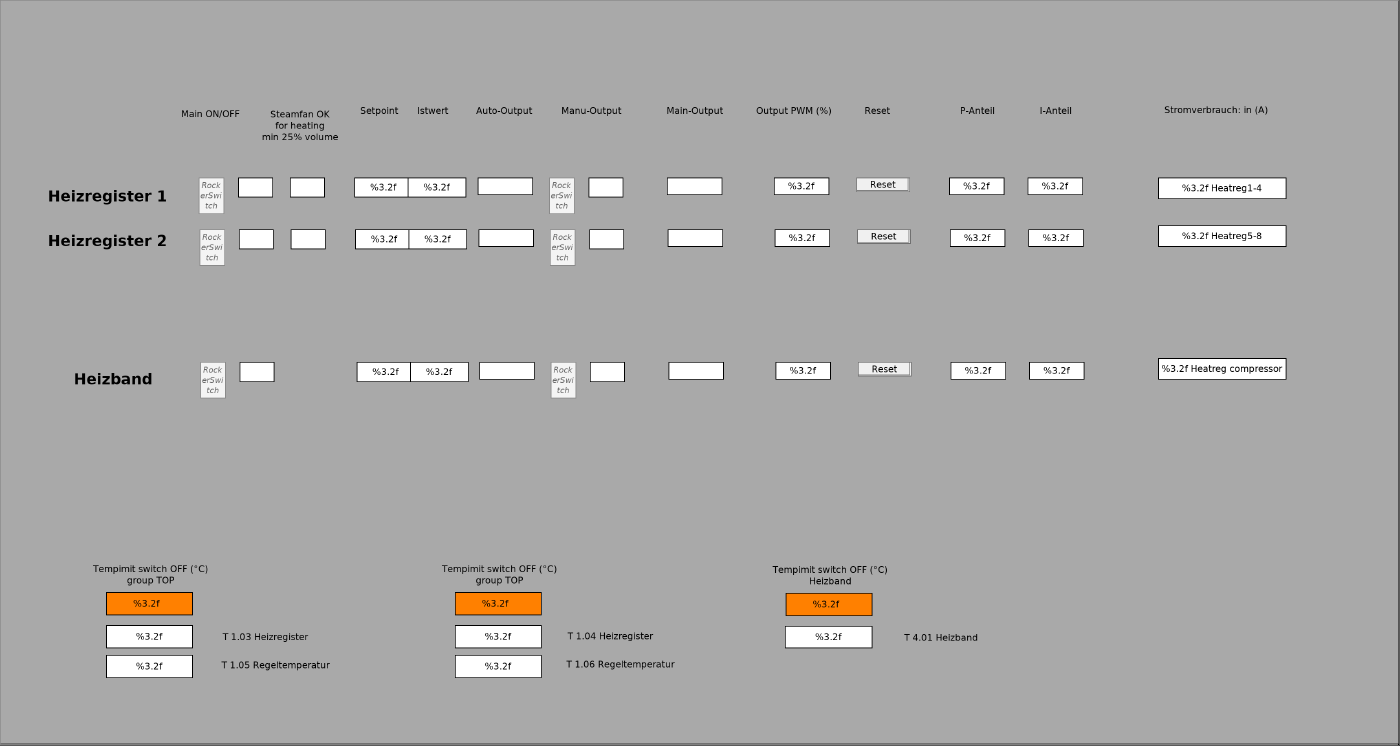
VISUALIZATION Heatreg  // 1782x950
    Rectangle (451,226 74x25), "%3.2f", tooltip "Durchmesser in mm eingeben", text variable: GVL.fSetpointValue1
        OnMouseDown: write the text variable via VisuDialogs.Numpad, min 0, max 150
    Rectangle (596,126 92x30), "Auto-Output"
    Rectangle (707,126 92x30), "Manu-Output"
    Rectangle (839,126 92x30), "Main-Output"
    Rectangle (437,126 92x30), "Setpoint"
    Rectangle (609,292 70x22), colour toggle: GVL.bAuto_Heat_REG2_CTRL
    Rectangle (850,292 70x22), colour toggle: GVL.HEAT_Reg_2_OUT
    Rectangle (608,226 70x22), colour toggle: GVL.bAuto_Heat_REG1_CTRL
    Rectangle (849,226 70x22), colour toggle: GVL.HEAT_Reg_1_OUT
    Rectangle (951,126 116x30), "Output PWM (%)"
    Rectangle (986,292 70x22), "%3.2f", text variable: fPWMDutyCycle2
    Rectangle (985,226 70x22), "%3.2f", text variable: fPWMDutyCycle1
    Rectangle (610,461 70x22), colour toggle: GVL.bAuto_Heat_REG3_CTRL
    Rectangle (851,461 70x22), colour toggle: GVL.HEAT_Reg_3_OUT
    Rectangle (987,461 70x22), "%3.2f", text variable: fPWMDutyCycle3
    Rectangle (1473,124 150x32), "Stromverbrauch: in (A)"
    Rectangle (750,292 44x25), colour toggle: GVL.bManuHeat_REG2_CTRL
    Rectangle (749,226 44x25), colour toggle: GVL.bManuHeat_REG1_CTRL
    Rectangle (751,461 44x25), colour toggle: GVL.bManuHeat_REG3_CTRL
    Rectangle (135,754 110x29), "%3.2f", tooltip "Durchmesser in mm eingeben", text variable: GVL.T_Limit_Heatreg_top
        OnMouseDown: write the text variable via VisuDialogs.Numpad, min 0, max 300
    Rectangle (107,718 170x28), "Tempimit switch OFF (°C) group TOP"
    Rectangle (135,796 110x29), "%3.2f", tooltip "Durchmesser in mm eingeben", text variable: GVL.T_HE_Einduesung_Oben_Visu
    Rectangle (135,834 110x29), "%3.2f", tooltip "Durchmesser in mm eingeben", text variable: GVL.T_Einduesung_Oben_Visu
    Rectangle (265,798 146x26), "T 1.03 Heizregister"
    Rectangle (265,834 172x26), "T 1.05 Regeltemperatur"
    Rectangle (579,754 110x29), "%3.2f", tooltip "Durchmesser in mm eingeben", text variable: GVL.T_Limit_Heatreg_bottom
        OnMouseDown: write the text variable via VisuDialogs.Numpad, min 0, max 300
    Rectangle (551,718 170x28), "Tempimit switch OFF (°C) group TOP"
    Rectangle (579,796 110x29), "%3.2f", tooltip "Durchmesser in mm eingeben", text variable: GVL.T_HE_Einduesung_Unten_Visu
    Rectangle (579,834 110x29), "%3.2f", tooltip "Durchmesser in mm eingeben", text variable: GVL.T_Einduesung_Unten_Visu
    Rectangle (1780,0 2x950)
    Rectangle (0,947 1780x3)
    RockerSwitch (699,226 32x46), variable: GVL.bManuHeat_REG1_CTRL, behaviour: TOGGLE, style: Switch-RockerSwitch-Gray
    RockerSwitch (700,292 32x46), variable: GVL.bManuHeat_REG2_CTRL, behaviour: TOGGLE, style: Switch-RockerSwitch-Gray
    RockerSwitch (701,461 32x46), variable: GVL.bManuHeat_REG3_CTRL, behaviour: TOGGLE, style: Switch-RockerSwitch-Gray
    Rectangle (452,292 74x25), "%3.2f", tooltip "Durchmesser in mm eingeben", text variable: GVL.fSetpointValue2
        OnMouseDown: write the text variable via VisuDialogs.Numpad, min 0, max 150
    Rectangle (454,461 74x25), "%3.2f", tooltip "Durchmesser in mm eingeben", text variable: GVL.fSetpointValue3
        OnMouseDown: write the text variable via VisuDialogs.Numpad, min 0, max 150
    Rectangle (1071,126 92x30), "Reset"
    Button (1092,461 68x18), "Reset"
        tap Reset_heatreg_compressor
    Button (1090,226 68x18), "Reset"
        tap Reset_heatreg_top
    Button (1091,292 68x18), "Reset"
        tap Reset_heatreg_bottom
    Rectangle (370,292 44x25), colour toggle: OK_For_HEAT_WHILE_FAN_IS_ON
    Rectangle (369,226 44x25), colour toggle: OK_For_HEAT_WHILE_FAN_IS_ON
    Rectangle (328,132 108x56), "Steamfan OK for heating min 25% volume"
    Rectangle (304,292 44x25), colour toggle: bManuHeat_REG2_switch_ON
    Rectangle (303,226 44x25), colour toggle: bManuHeat_REG1_switch_ON
    Rectangle (305,461 44x25), colour toggle: bManuHeat_REG3_switch_ON
    RockerSwitch (253,226 32x46), variable: bManuHeat_REG1_switch_ON, behaviour: TOGGLE, style: Switch-RockerSwitch-Gray
    RockerSwitch (254,292 32x46), variable: bManuHeat_REG2_switch_ON, behaviour: TOGGLE, style: Switch-RockerSwitch-Gray
    RockerSwitch (255,461 32x46), variable: bManuHeat_REG3_switch_ON, behaviour: TOGGLE, style: Switch-RockerSwitch-Gray
    Rectangle (222,130 92x30), "Main ON/OFF"
    Rectangle (1198,126 92x30), "P-Anteil"
    Rectangle (1209,292 70x22), "%3.2f", text variable: fKP_Controller_Heatmatt2
        OnMouseDown: write the text variable via VisuDialogs.Numpad, min 0, max 1000
    Rectangle (1208,226 70x22), "%3.2f", text variable: fKP_Controller_Heatmatt1
        OnMouseDown: write the text variable via VisuDialogs.Numpad, min 0, max 1000
    Rectangle (1210,461 70x22), "%3.2f", text variable: fKP_Controller_Heatmatt3
        OnMouseDown: write the text variable via VisuDialogs.Numpad, min 0, max 1000
    Rectangle (1298,126 92x30), "I-Anteil"
    Rectangle (1309,292 70x22), "%3.2f", text variable: fKI_Controller_Heatmatt2
        OnMouseDown: write the text variable via VisuDialogs.Numpad, min 0, max 1000
    Rectangle (1308,226 70x22), "%3.2f", text variable: fKI_Controller_Heatmatt1
        OnMouseDown: write the text variable via VisuDialogs.Numpad, min 0, max 1000
    Rectangle (1310,461 70x22), "%3.2f", text variable: fKI_Controller_Heatmatt3
        OnMouseDown: write the text variable via VisuDialogs.Numpad, min 0, max 1000
    Rectangle (40,235 194x30), "Heizregister 1"
    Rectangle (40,292 194x30), "Heizregister 2"
    Rectangle (47,468 194x30), "Heizband"
    Rectangle (704,797 146x26), "T 1.04 Heizregister"
    Rectangle (704,833 172x26), "T 1.06 Regeltemperatur"
    Rectangle (519,226 74x25), "%3.2f", tooltip "Durchmesser in mm eingeben", text variable: GVL.T_Einduesung_Oben_Visu
    Rectangle (505,126 92x30), "Istwert"
    Rectangle (520,292 74x25), "%3.2f", tooltip "Durchmesser in mm eingeben", text variable: GVL.T_Einduesung_Unten_Visu
    Rectangle (522,461 74x25), "%3.2f", tooltip "Durchmesser in mm eingeben", text variable: T_Komp_Gehaeuse_Visu
    Rectangle (999,797 111x28), "%3.2f", tooltip "Durchmesser in mm eingeben", text variable: T_Komp_Gehaeuse_Visu
    Rectangle (1000,755 110x29), "%3.2f", tooltip "Durchmesser in mm eingeben", text variable: T_Limit_Heatreg3
        OnMouseDown: write the text variable via VisuDialogs.Numpad, min 0, max 300
    Rectangle (972,719 170x28), "Tempimit switch OFF (°C) Heizband"
    Rectangle (1125,799 146x26), "T 4.01 Heizband"
    Rectangle (1474,226 163x27), "%3.2f Heatreg1-4", tooltip "Durchmesser in mm eingeben", text variable: Current_OUT_Heatreg_1_TO_4
    Rectangle (1474,287 163x27), "%3.2f Heatreg5-8", tooltip "Durchmesser in mm eingeben", text variable: Current_OUT_Heatreg_5_TO_8
    Rectangle (1474,456 163x27), "%3.2f Heatreg compressor", tooltip "Durchmesser in mm eingeben", text variable: Current_OUT_Heatreg_Compressor
END_VISUALIZATION

(* stored: Version 1.1.0.1, ProductVersion 3.1.4024.3
   Visu Heatreg: Id {41f78d3a-a824-4dde-b9d8-d22bf7d9aae9} *)
